TYPE ST_HmiRow :
STRUCT
    nIndex : UINT;
    sName : STRING(40);
    lrValue : LREAL;
    bEnabled : BOOL;
    sUnit : STRING(16);
    sSource : STRING(16);
END_STRUCT
END_TYPE

(* stored: Version 1.1.0.1
   DUT ST_HmiRow: Id {a7df6fcf-7a89-46b1-a1aa-1e58d50bfca8} *)
